Universal Robots PolyScope program: 123.urp

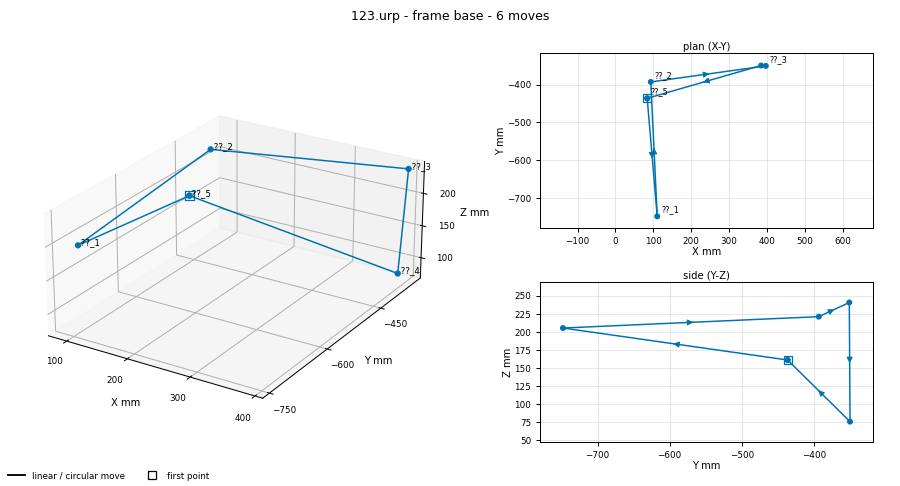
[picture p0: tool path of 123.urp in frame base, 6 of 6 moves have a stored position in this frame; points joined in program order, loops and branches not executed]
Program 123 (installation=20240827 directory=/programs/collection createdIn=5.15.1 lastSavedIn=5.15.1 robotSerialNumber=20245500285)
Calibrated DH parameters: a=[0.000097, -0.210459, -0.026602, 0.000137, 0.000078, 0]; d=[0.162601, 254.180657, -54.076236, -199.970743, 0.099615, 0.099684]; alpha=[1.569796, -0.001455, 0.001957, 1.570525, -1.571561, 0]; deltaTheta=[0, -1.053331, 8.839472, -1.50296, 0.000002, 0]
InitVariablesNode
Robot Program (runOnlyOnce=false)
  SuppressedNode
    MoveJ speed 60 deg/s, acceleration 80 deg/s^2 (useActiveTCP=true) feature=Base
      Waypoint 路点_5: TCP in base x=83.88 y=-436.387 z=161.231 mm, rx=-1.9721 ry=-1.9405 rz=-0.512 rad; joints [84.13, -76.56, 92.844, -78.269, -91.203, 85.541] deg; TCP offset x=-0.17 y=0 z=192.95 mm, rx=0 ry=0 rz=0 rad
      Waypoint 路点_1: TCP in base x=110.372 y=-747.932 z=205.564 mm, rx=2.118 ry=2.1976 rz=-0.0783 rad; joints [87.392, -58.175, 63.597, -101.028, -88.173, 85.568] deg
      Waypoint 路点_2: TCP in base x=93.347 y=-393.146 z=221.344 mm, rx=2.2182 ry=2.1468 rz=0.1116 rad; joints [80.168, -104.699, 113.272, -97.057, -85.108, 82.128] deg
      Waypoint 路点_3: TCP in base x=396.924 y=-350.898 z=240.978 mm, rx=2.1925 ry=2.1616 rz=0.1271 rad; joints [120.727, -89.179, 97.93, -101.024, -84.588, 121.819] deg
      Waypoint 路点_4: TCP in base x=384.441 y=-349.869 z=75.744 mm, rx=2.2342 ry=2.1982 rz=0.0936 rad; joints [120.73, -80.387, 113.334, -122.513, -86.643, 121.814] deg
      Waypoint 路点_5: TCP in base x=83.88 y=-436.387 z=161.231 mm, rx=-1.9721 ry=-1.9405 rz=-0.512 rad; joints [84.13, -76.56, 92.844, -78.269, -91.203, 85.541] deg
      Popup Message (haltProgram=false message=211 inputType=Text)
  MoveL speed 3000 mm/s, acceleration 2500 mm/s^2 (useActiveTCP=true) feature=Base
    Waypoint 路点_5: TCP in base x=83.88 y=-436.387 z=161.231 mm, rx=-1.9721 ry=-1.9405 rz=-0.512 rad; joints [84.13, -76.56, 92.844, -78.269, -91.203, 85.541] deg
    Waypoint 路点_1: TCP in base x=110.372 y=-747.932 z=205.564 mm, rx=2.118 ry=2.1976 rz=-0.0783 rad; joints [87.392, -58.175, 63.597, -101.028, -88.173, 85.568] deg
    Waypoint 路点_2: TCP in base x=93.347 y=-393.146 z=221.344 mm, rx=2.2182 ry=2.1468 rz=0.1116 rad; joints [80.168, -104.699, 113.272, -97.057, -85.108, 82.128] deg
    Waypoint 路点_3: TCP in base x=396.924 y=-350.898 z=240.978 mm, rx=2.1925 ry=2.1616 rz=0.1271 rad; joints [120.727, -89.179, 97.93, -101.024, -84.588, 121.819] deg
    Waypoint 路点_4: TCP in base x=384.441 y=-349.869 z=75.744 mm, rx=2.2342 ry=2.1982 rz=0.0936 rad; joints [120.73, -80.387, 113.334, -122.513, -86.643, 121.814] deg
    Waypoint 路点_5: TCP in base x=83.88 y=-436.387 z=161.231 mm, rx=-1.9721 ry=-1.9405 rz=-0.512 rad; joints [84.13, -76.56, 92.844, -78.269, -91.203, 85.541] deg
    Popup Message (haltProgram=false message=211 inputType=Text)
